Universal Robots PolyScope program: 9-set.urp

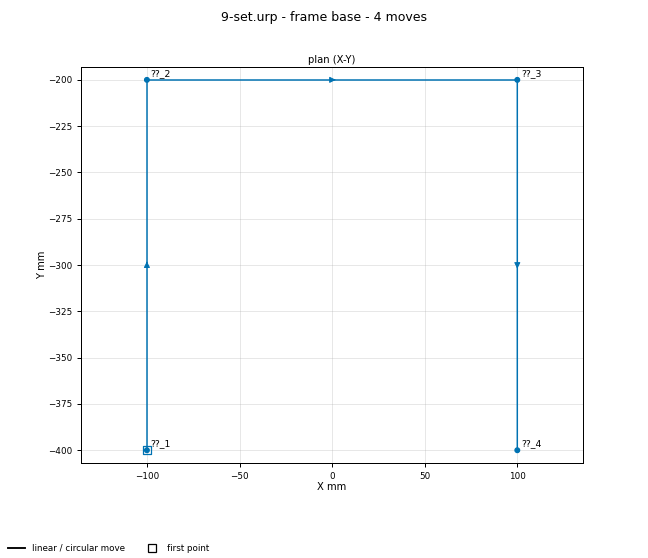
[picture p0: tool path of 9-set.urp in frame base, 4 of 4 moves have a stored position in this frame; points joined in program order, loops and branches not executed]
ProgramRoot directory=/home/ur/ursim-3.1/programs/basic training/9-set; kinematics=(a=[0, -0.425, -0.39225, 0, 0, 0], d=[0.08916, 0, 0, 0.10915, 0.09465, 0.0823], alpha=[1.5708, 0, 0, 1.5708, -1.5708, 0], deltaTheta=[0, 0, 0, 0, 0, 0], status=notInitialized); lastSavedInVersion=(project__name=Polyscope, major__version=3, minor__version=1, svn__revision=17195, build__date=Mar 11 2015, 13:02:28); name=9-set; programVersion=(project__name=Polyscope, major__version=3, minor__version=1, svn__revision=17195, build__date=Mar 11 2015, 13:02:28); robotEnvironmentFileName=default; serialNumberRobot=2014350001
  MainProgram cartesianAcceleration=1.2; cartesianSpeed=0.25; jointAcceleration=1.3962634015954636; jointSpeed=1.0471975511965976; sharedProcessMoveBlendRadius=0.025; motionType=JOINT_SPACE
    Move cartesianAcceleration=1.2; cartesianSpeed=0.25; jointAcceleration=1.3962634015954636; jointSpeed=1.0471975511965976; sharedProcessMoveBlendRadius=0.025; motionType=CARTESIAN_SPACE
      Waypoint blendRadius=0.05; cartesianAcceleration=1.2; cartesianSpeed=0.25; jointAcceleration=1.3962634015954636; jointSpeed=1.0471975511965976; nextMotionTime=2.0; stoppoint=true; useSharedBlendParameter=true; useSharedParameters=true; outputFlangePose=(pos=(x=-0.10000000065989616, y=-0.40000000104212996, z=0.1999999982306596), rot=(x=-0.0012209830283997337, y=3.116276481240887, z=0.0388919161681283)); position=TCP in base x=-100 y=-400 z=200 mm, rx=-0.0012 ry=3.1163 rz=0.0389 rad; joints [-88.988, -88.3, -127.491, -55.614, 91.461, 0.95] deg; positionType=FIXED_POSITION; waypointPoseInFeatureCoordinates=(pos=(x=-0.09999996819589951, y=-0.40000005265404437, z=0.1999999632555712), rot=(x=-0.0012210995530369398, y=3.1162764787073427, z=0.0388923209577584)); name=路点_1
      Set 
      Waypoint blendRadius=0.05; cartesianAcceleration=1.2; cartesianSpeed=0.25; jointAcceleration=1.3962634015954636; jointSpeed=1.0471975511965976; nextMotionTime=2.0; stoppoint=true; useSharedBlendParameter=true; useSharedParameters=true; outputFlangePose=(pos=(x=-0.09999996819589557, y=-0.2000000004084386, z=0.1999999632555922), rot=(x=-0.0012210995530455748, y=3.1162764787073587, z=0.03889232095787024)); position=TCP in base x=-100 y=-200 z=200 mm, rx=-0.0012 ry=3.1163 rz=0.0389 rad; joints [-87.972, -51.697, -148.925, -70.758, 91.486, 1.966] deg; positionType=FIXED_POSITION; waypointPoseInFeatureCoordinates=(pos=(x=-0.1000000033773473, y=-0.1999999639802142, z=0.1999999879203018), rot=(x=-0.0012208534573265933, y=3.1162765026745864, z=0.03889211050910507)); name=路点_2
      Waypoint blendRadius=0.05; cartesianAcceleration=1.2; cartesianSpeed=0.25; jointAcceleration=1.3962634015954636; jointSpeed=1.0471975511965976; nextMotionTime=2.0; stoppoint=true; useSharedBlendParameter=true; useSharedParameters=true; outputFlangePose=(pos=(x=0.0999999994889211, y=-0.1999999639801891, z=0.19999998792032553), rot=(x=-0.001220853457196563, y=3.1162765026745523, z=0.03889211050897391)); position=TCP in base x=100 y=-200 z=200 mm, rx=-0.0012 ry=3.1163 rz=0.0389 rad; joints [-35.055, -51.443, -149.443, -68.76, 91.996, 54.906] deg; positionType=FIXED_POSITION; waypointPoseInFeatureCoordinates=(pos=(x=0.10000003093004557, y=-0.19999997679952106, z=0.20000002024915683), rot=(x=-0.0012209058668588384, y=3.1162765360370175, z=0.03889203442947606)); name=路点_3
      Waypoint blendRadius=0.05; cartesianAcceleration=1.2; cartesianSpeed=0.25; jointAcceleration=1.3962634015954636; jointSpeed=1.0471975511965976; nextMotionTime=2.0; stoppoint=true; useSharedBlendParameter=true; useSharedParameters=true; outputFlangePose=(pos=(x=0.10000003093003211, y=-0.39999999959145743, z=0.2000000202491417), rot=(x=-0.001220905866926126, y=3.116276536037035, z=0.03889203442951857)); position=TCP in base x=100 y=-400 z=200 mm, rx=-0.0012 ry=3.1163 rz=0.0389 rad; joints [-61.016, -88.295, -127.75, -54.511, 91.949, 28.93] deg; positionType=FIXED_POSITION; waypointPoseInFeatureCoordinates=(pos=(x=0.10000008984723645, y=-0.39999992995872546, z=0.19999983963652107), rot=(x=-0.0012212291743970486, y=3.116276825726508, z=0.038892683103293996)); name=路点_4
      Set 
